Fanuc TP program (LS listing): timer.ls

/PROG  TIMER	  Macro
/ATTR
OWNER		= MNEDITOR;
COMMENT		= "CYCLE TIME";
PROG_SIZE	= 243;
CREATE		= DATE 26-02-10  TIME 10:54:34;
MODIFIED	= DATE 26-02-10  TIME 10:55:22;
FILE_NAME	= ;
VERSION		= 0;
LINE_COUNT	= 10;
MEMORY_SIZE	= 575;
PROTECT		= READ_WRITE;
TCD:  STACK_SIZE	= 0,
      TASK_PRIORITY	= 50,
      TIME_SLICE	= 0,
      BUSY_LAMP_OFF	= 0,
      ABORT_REQUEST	= 0,
      PAUSE_REQUEST	= 0;
DEFAULT_GROUP	= 1,*,*,*,*;
CONTROL_CODE	= 00000000 00000000;
LOCAL_REGISTERS	= 0,0,0;
/APPL

AUTO_SINGULARITY_HEADER;
  ENABLE_SINGULARITY_AVOIDANCE   : TRUE;
/MN
   1:   ;
   2:   ;
   3:   ;
   4:   ;
   5:   ;
   6:   ;
   7:   ;
   8:   ;
   9:   ;
  10:   ;
/POS
/END
